TYPE ST_AteqCommands :
STRUCT

    (* Byte 0 - 00h *)
    bReset                     : BOOL; // Bit 0
    bStart                     : BOOL; // Bit 1
    bSpecialCycle              : BOOL; // Bit 2
    bProgramSelect             : BOOL; // Bit 3
    bReadFifoResults           : BOOL; // Bit 4
    bReadParameters            : BOOL; // Bit 5
    bWriteParameters           : BOOL; // Bit 6
    bResetFifo                 : BOOL; // Bit 7

    (* Byte 1 - 01h *)
    bReadInstrumentConfig      : BOOL; // Bit 0
    bReadConfig	               : BOOL; // Bit 1
    bReadFunctionBits          : BOOL; // Bit 2
    bWriteExtMenu              : BOOL; // Bit 3
    bWriteFunctionBits         : BOOL; // Bit 4
    bReadProgramName           : BOOL; // Bit 5
    bWriteProgramName          : BOOL; // Bit 6
    bReadLastResult            : BOOL; // Bit 7

END_STRUCT
END_TYPE

(* stored: Version 1.1.0.1, ProductVersion 3.1.4024.15
   DUT ST_AteqCommands: Id {b1936584-ffcc-4a62-8179-6b1a04071057} *)
